(* Logix 5000 project; controller TP_EOL20161211 1769-L16ER-BB1B rev 20.12; software revision 20.01; part 2 of 2 *)
(* tags used below, declared in another part *)
   Cmd_VJOS_GJD : BOOL;
   Cmd_VJOS_GJF : BOOL;
   Cmd_VJOS_GJN : BOOL;
   Cmd_VJOS_GST : BOOL;
   Cmd_VJOS_OfflineRequest : BOOL;
   Cmd_VJOS_RunRequest : BOOL;
   Cmd_VJOS_ShutDownRequest : BOOL;
   Cmd_VJOS_ShuttingDownRequest : BOOL;
   Cmd_VJOS_SLA : BOOL;
   Cmd_VJOS_StartupRequest : BOOL;
   CO_Trigger : DINT;
   CO_VJCTUOS : COUNTER;
   Par_JobSelect : STRING;
   Par_VarData : STRING;
   Par_VJ_JobSelect : STRING;
   Sts_VJOS_CurrentJob : STRING;
   VJ_ACK : STRING;
   VJ_Blank : STRING;
   VJ_FieldData : STRING;
   VJ_FieldPos : INT;
   VJ_PLC01 : STRING;
   VJ_VarDataPOS : INT;
   VJOS_JobFieldDataErr : BOOL;
   VJOS_JobSLAErr : BOOL;
   VJOS_msgSeq : INT;
   VJOS_ReadTimer : TIMER[10];
   VJOS_Wrk_Jobassign : STRING;
   VOS_SKT_Client_AOI : SKT_TCP_CLIENT_AOI;
   wrk_Concat : STRING;
   wrk_ConcatSLA : STRING;
   wrk_GJD : STRING;
   wrk_GJF : STRING;
   wrk_GJN : STRING;
   wrk_GST : STRING;
   wrk_SLA : STRING;
   wrk_State : STRING;
   wrk_StateCmd : STRING;
   nc_CO_Cmd : UDT_EOLPlus;
   VOS_SKT_Client_Connect_MSG : MESSAGE;
   VOS_SKT_Client_Create_MSG : MESSAGE;
   VOS_SKT_Client_DATA : SKT_DATA_CLIENT;
   VOS_SKT_Client_Delete_MSG : MESSAGE;
   VOS_SKT_Client_Port : DINT;
   VOS_SKT_Client_Read_MSG : MESSAGE;
   VOS_SKT_Client_Write_MSG : MESSAGE;
   VOS_SKT_Delete_All_MSG : MESSAGE;
   VOS_SKT_Device_IP_Port_Server : STRING;
   VOS_SKT_MSG_PATH : STRING;
   VOS_SKT_String_recieved : STR_480;
   VOS_SKT_String_to_send : STR_480;
   VOS_SKT_Toggle : DINT;
(* Comm, continued *)

ROUTINE VideoJetOS   (* ladder *)
// 192.168.1.65
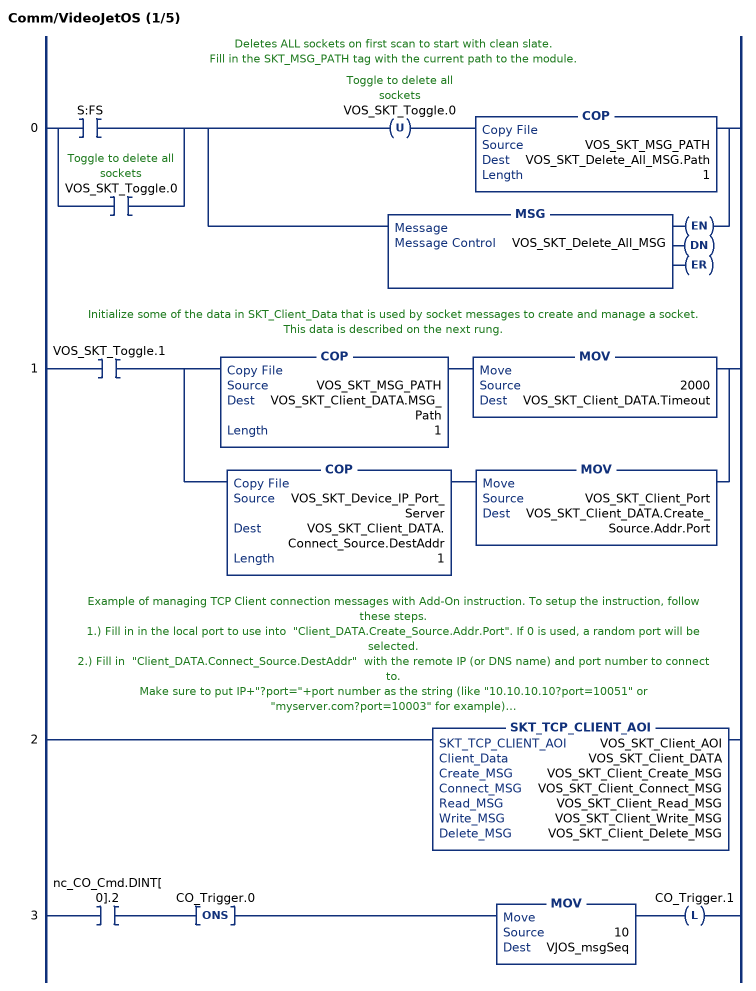
   // Deletes ALL sockets on first scan to start with clean slate.
   // Fill in the SKT_MSG_PATH tag with the current path to the module.
   0: [XIC(S:FS) ,XIC(VOS_SKT_Toggle.0) ][OTU(VOS_SKT_Toggle.0) COP(VOS_SKT_MSG_PATH,VOS_SKT_Delete_All_MSG.Path,1) ,MSG(VOS_SKT_Delete_All_MSG) ];
   // Initialize some of the data in SKT_Client_Data that is used by socket messages to create and manage a socket.
   // This data is described on the next rung.
   1: XIC(VOS_SKT_Toggle.1)[COP(VOS_SKT_MSG_PATH,VOS_SKT_Client_DATA.MSG_Path,1) MOV(2000,VOS_SKT_Client_DATA.Timeout) ,COP(VOS_SKT_Device_IP_Port_Server,VOS_SKT_Client_DATA.Connect_Source.DestAddr,1) MOV(VOS_SKT_Client_Port,VOS_SKT_Client_DATA.Create_Source.Addr.Port) ];
   // Example of managing TCP Client connection messages with Add-On instruction. To setup the instruction, follow these steps.
   // 1.) Fill in in the local port to use into  "Client_DATA.Create_Source.Addr.Port". If 0 is used, a random port will be selected.
   // 2.) Fill in  "Client_DATA.Connect_Source.DestAddr"  with the remote IP (or DNS name) and port number to connect to.
   // Make sure to put IP+"?port="+port number as the string (like "10.10.10.10?port=10051" or "myserver.com?port=10003" for example).
   // 3.) Fill in the path to the module in the SKT_MSG_PATH tag (the path will look like "$01$03" for slot 3, for example).
   // 4.) To start or stop the client connection, set or clear the Enable_Socket respectively.
   // 5.) If trying to trap error for troubleshooting the connection, the set the Stop_on_Error bit on the instruction. If there is an error, the instruction will clear the Stop_on_Errorwhen a message errors.
   // The SC status bit means trying to connect. The SO status bit means Socket Connected and open. The ER bit means a message ERrored.
   // When the DR bit is set by the instruction, then there is string data that arrived from the socket. Copy the string data if desired and clear the DR bit to get new data.
   // When data needs to be sent by the application, fill in the string data into "Client_DATA.Write_Source.Buffer", then set the WD bit. The instruction will clear the WD bit when the data is written.
   // Modify the rung branches to suit the application.
   2: SKT_TCP_CLIENT_AOI(VOS_SKT_Client_AOI,VOS_SKT_Client_DATA,VOS_SKT_Client_Create_MSG,VOS_SKT_Client_Connect_MSG,VOS_SKT_Client_Read_MSG,VOS_SKT_Client_Write_MSG,VOS_SKT_Client_Delete_MSG);
   3: XIC(nc_CO_Cmd.DINT[0].2)ONS(CO_Trigger.0)MOV(10,VJOS_msgSeq)OTL(CO_Trigger.1);
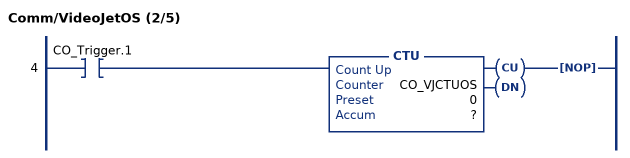
   4: XIC(CO_Trigger.1)CTU(CO_VJCTUOS,?,?)NOP();
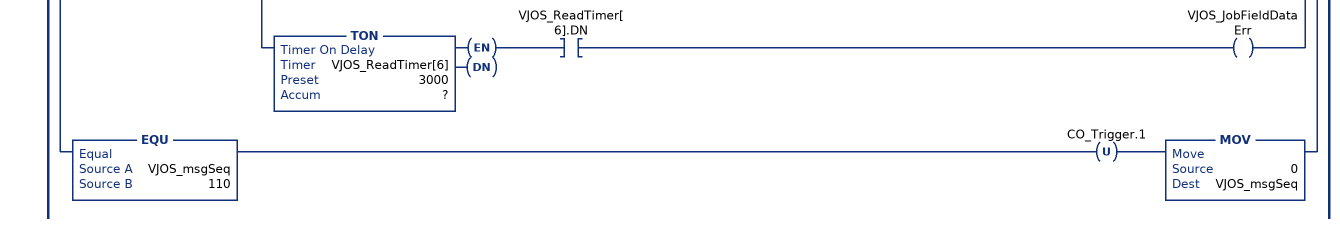
   5: [EQU(VJOS_msgSeq,10) [XIC(VOS_SKT_Client_AOI.DR) TON(VJOS_ReadTimer[0],?,?) XIC(VJOS_ReadTimer[0].DN) OTL(VOS_SKT_Toggle.3) ,XIO(VOS_SKT_Client_AOI.DR) TON(VJOS_ReadTimer[1],?,?) XIC(VJOS_ReadTimer[1].DN) MOV(20,VJOS_msgSeq) ] ,EQU(VJOS_msgSeq,20) NEQ(VJ_Blank,Par_VJ_JobSelect) NEQ(VJ_Blank,Par_VarData) OTL(Cmd_VJOS_SLA) MOV(25,VJOS_msgSeq) ,EQU(VJOS_msgSeq,25) OTL(VOS_SKT_Toggle.2) XIC(VOS_SKT_Client_AOI.WD) MOV(30,VJOS_msgSeq) ,EQU(VJOS_msgSeq,30) TON(VJOS_ReadTimer[2],?,?) XIC(VJOS_ReadTimer[2].DN) XIC(VOS_SKT_Client_AOI.DR) OTL(VOS_SKT_Toggle.3) MOV(40,VJOS_msgSeq) ,EQU(VJOS_msgSeq,40) EQU(VJ_ACK,VOS_SKT_String_recieved) OTL(VOS_SKT_Toggle.3) MOV(50,VJOS_msgSeq) ,EQU(VJOS_msgSeq,50) OTL(Cmd_VJOS_GJN) MOV(55,VJOS_msgSeq) ,EQU(VJOS_msgSeq,55) OTL(VOS_SKT_Toggle.2) XIC(VOS_SKT_Client_AOI.WD) MOV(60,VJOS_msgSeq) ,EQU(VJOS_msgSeq,60) TON(VJOS_ReadTimer[3],?,?) XIC(VJOS_ReadTimer[3].DN) XIC(VOS_SKT_Client_AOI.DR) OTL(VOS_SKT_Toggle.3) MOV(70,VJOS_msgSeq) ,EQU(VJOS_msgSeq,70) [MID(VOS_SKT_String_recieved,8,5,Sts_VJOS_CurrentJob) EQU(Sts_VJOS_CurrentJob,Par_VJ_JobSelect) MOV(80,VJOS_msgSeq) ,TON(VJOS_ReadTimer[5],?,?) XIC(VJOS_ReadTimer[5].DN) OTE(VJOS_JobSLAErr) ] ,EQU(VJOS_msgSeq,80) OTL(Cmd_VJOS_GJD) MOV(85,VJOS_msgSeq) ,EQU(VJOS_msgSeq,85) OTL(VOS_SKT_Toggle.2) XIC(VOS_SKT_Client_AOI.WD) MOV(90,VJOS_msgSeq) ,EQU(VJOS_msgSeq,90) TON(VJOS_ReadTimer[4],?,?) XIC(VJOS_ReadTimer[4].DN) XIC(VOS_SKT_Client_AOI.DR) OTL(VOS_SKT_Toggle.3) MOV(100,VJOS_msgSeq) ,EQU(VJOS_msgSeq,100) [FIND(VOS_SKT_String_recieved,VJ_PLC01,5,VJ_FieldPos) ADD(VJ_FieldPos,6,VJ_VarDataPOS) MID(VOS_SKT_String_recieved,10,VJ_VarDataPOS,VJ_FieldData) EQU(VJ_FieldData,Par_VarData) MOV(110,VJOS_msgSeq) ,TON(VJOS_ReadTimer[6],?,?) XIC(VJOS_ReadTimer[6].DN) OTE(VJOS_JobFieldDataErr) ] ,EQU(VJOS_msgSeq,110) OTU(CO_Trigger.1) MOV(0,VJOS_msgSeq) ];
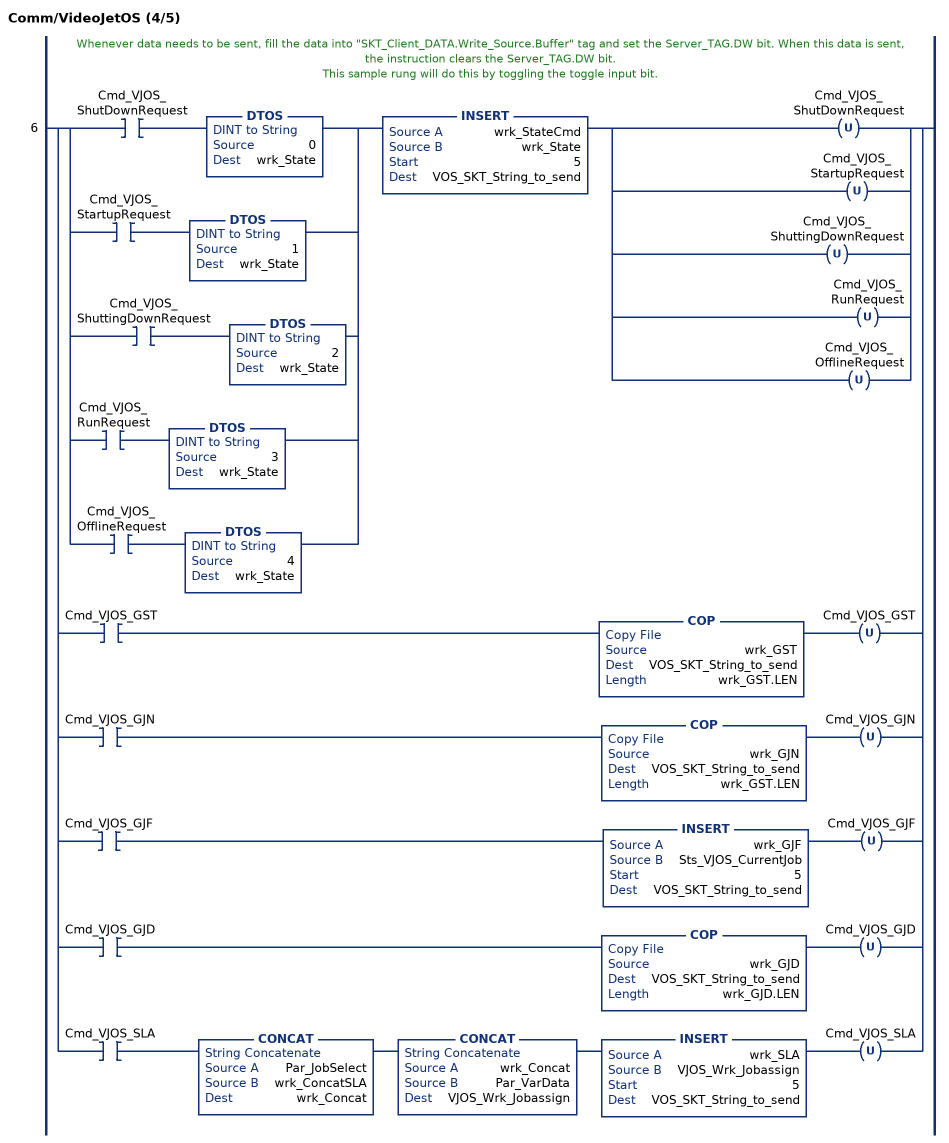
   // Whenever data needs to be sent, fill the data into "SKT_Client_DATA.Write_Source.Buffer" tag and set the Server_TAG.DW bit. When this data is sent, the instruction clears the Server_TAG.DW bit.
   // This sample rung will do this by toggling the toggle input bit.
   6: [[XIC(Cmd_VJOS_ShutDownRequest) DTOS(0,wrk_State) ,XIC(Cmd_VJOS_StartupRequest) DTOS(1,wrk_State) ,XIC(Cmd_VJOS_ShuttingDownRequest) DTOS(2,wrk_State) ,XIC(Cmd_VJOS_RunRequest) DTOS(3,wrk_State) ,XIC(Cmd_VJOS_OfflineRequest) DTOS(4,wrk_State) ] INSERT(wrk_StateCmd,wrk_State,5,VOS_SKT_String_to_send) [OTU(Cmd_VJOS_ShutDownRequest) ,OTU(Cmd_VJOS_StartupRequest) ,OTU(Cmd_VJOS_ShuttingDownRequest) ,OTU(Cmd_VJOS_RunRequest) ,OTU(Cmd_VJOS_OfflineRequest) ] ,XIC(Cmd_VJOS_GST) COP(wrk_GST,VOS_SKT_String_to_send,wrk_GST.LEN) OTU(Cmd_VJOS_GST) ,XIC(Cmd_VJOS_GJN) COP(wrk_GJN,VOS_SKT_String_to_send,wrk_GST.LEN) OTU(Cmd_VJOS_GJN) ,XIC(Cmd_VJOS_GJF) INSERT(wrk_GJF,Sts_VJOS_CurrentJob,5,VOS_SKT_String_to_send) OTU(Cmd_VJOS_GJF) ,XIC(Cmd_VJOS_GJD) COP(wrk_GJD,VOS_SKT_String_to_send,wrk_GJD.LEN) OTU(Cmd_VJOS_GJD) ,XIC(Cmd_VJOS_SLA) CONCAT(Par_JobSelect,wrk_ConcatSLA,wrk_Concat) CONCAT(wrk_Concat,Par_VarData,VJOS_Wrk_Jobassign) INSERT(wrk_SLA,VJOS_Wrk_Jobassign,5,VOS_SKT_String_to_send) OTU(Cmd_VJOS_SLA) ];
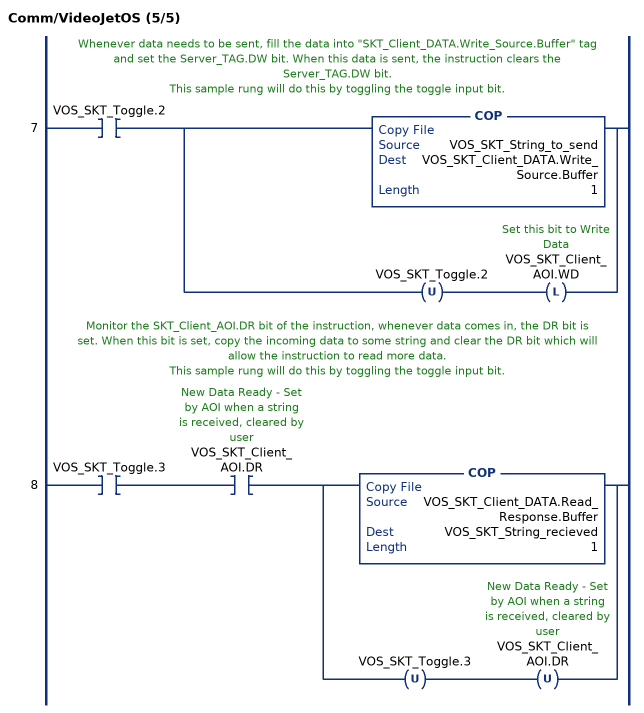
   // Whenever data needs to be sent, fill the data into "SKT_Client_DATA.Write_Source.Buffer" tag and set the Server_TAG.DW bit. When this data is sent, the instruction clears the Server_TAG.DW bit.
   // This sample rung will do this by toggling the toggle input bit.
   7: XIC(VOS_SKT_Toggle.2)[COP(VOS_SKT_String_to_send,VOS_SKT_Client_DATA.Write_Source.Buffer,1) ,OTU(VOS_SKT_Toggle.2) OTL(VOS_SKT_Client_AOI.WD) ];
   // Monitor the SKT_Client_AOI.DR bit of the instruction, whenever data comes in, the DR bit is set. When this bit is set, copy the incoming data to some string and clear the DR bit which will allow the instruction to read more data.
   // This sample rung will do this by toggling the toggle input bit.
   8: XIC(VOS_SKT_Toggle.3)XIC(VOS_SKT_Client_AOI.DR)[COP(VOS_SKT_Client_DATA.Read_Response.Buffer,VOS_SKT_String_recieved,1) ,OTU(VOS_SKT_Toggle.3) OTU(VOS_SKT_Client_AOI.DR) ];
END_ROUTINE
END_PROGRAM
